TYPE AX5000_P_0361 :
STRUCT
	Actual_lenght:UINT;
	Max_lenght:UINT;
	Parameter_set_configuration:ARRAY[0..34] OF UINT;
END_STRUCT
END_TYPE

(* stored: Version 1.1.0.1, ProductVersion 3.1.4024.3
   DUT AX5000_P_0361: Id {a11aa558-7d36-4df2-b92f-fd455da267f7} *)
